FUNCTION sign : int
VAR_INPUT
	value : LREAL;
END_VAR
VAR
END_VAR

IF value > 0 THEN 
	sign := 1;
ELSIF value <  0 THEN
	sign :=-1;
ELSE 
	sign :=0;
END_IF

END_FUNCTION

(* stored: Version 1.1.0.1, ProductVersion 3.1.4024.12
   POU sign: Id {73314d4f-8960-4437-b969-7aac31f0a87d}, SpecialFunc None *)
